{attribute addProperty BoxType ""}
{attribute addProperty Id "_defaultSyncUnitTasks_F32BF96626032.50"}
{attribute addProperty CRC "592655343"}
{attribute addProperty SizeInBites "260"}
{attribute addProperty SizeInBytes "32.5"}
TYPE SyncUnits_235333EF :
STRUCT
	{attribute addProperty Name "_default"}
	_default : SyncUnitTasks_F32BF966;
END_STRUCT
END_TYPE

(* stored: Version 1.2.0.0, ProductVersion 3.1.4024.9
   DUT SyncUnits_235333EF: Id {590925a6-124f-0b9f-0bb2-ff4c46d57978} *)
